  MoveL (T20104) to (112.13, 109.45, 20.1) mm, rotated rx 180 ry 0 rz -180 deg; joints [1.817, 69.838, -35.399, 3.211, -34.481, -2.648]
  Call Extruder 0.01136
  MoveL (T20105) to (122.25, 109.45, 20.1) mm, rotated rx 180 ry 0 rz -180 deg; joints [1.817, 69.838, -35.399, 3.211, -34.481, -2.648]
  Call Extruder 0.00011
  MoveL (T20106) to (122.25, 109.35, 20.1) mm, rotated rx 180 ry 0 rz -180 deg; joints [1.817, 69.838, -35.399, 3.211, -34.481, -2.648]
  Call Extruder 0.01142
  MoveL (T20107) to (112.08, 109.35, 20.1) mm, rotated rx 180 ry 0 rz -180 deg; joints [1.416, 68.674, -33.212, 2.439, -35.486, -1.986]
  Call Extruder 0.00013
  MoveL (T20108) to (112.03, 109.25, 20.1) mm, rotated rx 180 ry 0 rz -180 deg; joints [1.416, 68.674, -33.212, 2.439, -35.486, -1.986]
  Call Extruder 0.01148
  MoveL (T20109) to (122.25, 109.25, 20.1) mm, rotated rx 180 ry 0 rz -180 deg; joints [1.416, 68.674, -33.212, 2.439, -35.486, -1.986]
  Call Extruder 0.00011
  MoveL (T20110) to (122.25, 109.15, 20.1) mm, rotated rx 180 ry 0 rz -180 deg; joints [1.417, 68.506, -32.897, 2.433, -35.633, -1.978]
  Call Extruder 0.01153
  MoveL (T20111) to (111.98, 109.15, 20.1) mm, rotated rx 180 ry 0 rz -180 deg; joints [1.417, 68.506, -32.897, 2.433, -35.633, -1.978]
  Call Extruder 0.00013
  MoveL (T20112) to (111.92, 109.05, 20.1) mm, rotated rx 180 ry 0 rz -180 deg; joints [1.819, 69.662, -35.069, 3.202, -34.636, -2.636]
  Call Extruder 0.01159
  MoveL (T20113) to (122.25, 109.05, 20.1) mm, rotated rx 180 ry 0 rz -180 deg; joints [1.819, 69.662, -35.069, 3.202, -34.636, -2.636]
  Call Extruder 0.00011
  MoveL (T20114) to (122.25, 108.95, 20.1) mm, rotated rx 180 ry 0 rz -180 deg; joints [1.819, 69.662, -35.069, 3.202, -34.636, -2.636]
  Call Extruder 0.01165
  MoveL (T20115) to (111.87, 108.95, 20.1) mm, rotated rx 180 ry 0 rz -180 deg; joints [1.821, 69.488, -34.741, 3.193, -34.789, -2.624]
  Call Extruder 0.00013
  MoveL (T20116) to (111.82, 108.85, 20.1) mm, rotated rx 180 ry 0 rz -180 deg; joints [1.821, 69.488, -34.741, 3.193, -34.789, -2.624]
  Call Extruder 0.01171
  MoveL (T20117) to (122.25, 108.85, 20.1) mm, rotated rx 180 ry 0 rz -180 deg; joints [1.419, 68.339, -32.584, 2.427, -35.78, -1.969]
  Call Extruder 0.00011
  MoveL (T20118) to (122.25, 108.75, 20.1) mm, rotated rx 180 ry 0 rz -180 deg; joints [1.419, 68.339, -32.584, 2.427, -35.78, -1.969]
  Call Extruder 0.01176
  MoveL (T20119) to (111.77, 108.75, 20.1) mm, rotated rx 180 ry 0 rz -180 deg; joints [1.42, 68.174, -32.273, 2.421, -35.925, -1.961]
  Call Extruder 0.00013
  MoveL (T20120) to (111.72, 108.65, 20.1) mm, rotated rx 180 ry 0 rz -180 deg; joints [1.42, 68.174, -32.273, 2.421, -35.925, -1.961]
  Call Extruder 0.01182
  MoveL (T20121) to (122.25, 108.65, 20.1) mm, rotated rx 180 ry 0 rz -180 deg; joints [1.42, 68.174, -32.273, 2.421, -35.925, -1.961]
  Call Extruder 0.00011
  MoveL (T20122) to (122.25, 108.55, 20.1) mm, rotated rx 180 ry 0 rz -180 deg; joints [1.823, 69.314, -34.415, 3.185, -34.941, -2.612]
  Call Extruder 0.01188
  MoveL (T20123) to (111.67, 108.55, 20.1) mm, rotated rx 180 ry 0 rz -180 deg; joints [1.823, 69.314, -34.415, 3.185, -34.941, -2.612]
  Call Extruder 0.00013
  MoveL (T20124) to (111.62, 108.45, 20.1) mm, rotated rx 180 ry 0 rz -180 deg; joints [1.823, 69.314, -34.415, 3.185, -34.941, -2.612]
  Call Extruder 0.01194
  MoveL (T20125) to (122.25, 108.45, 20.1) mm, rotated rx 180 ry 0 rz -180 deg; joints [1.825, 69.142, -34.092, 3.176, -35.092, -2.6]
  Call Extruder 0.00011
  MoveL (T20126) to (122.25, 108.35, 20.1) mm, rotated rx 180 ry 0 rz -180 deg; joints [1.825, 69.142, -34.092, 3.176, -35.092, -2.6]
  Call Extruder 0.01205
  MoveL (T20127) to (111.52, 108.35, 20.1) mm, rotated rx 180 ry 0 rz -180 deg; joints [1.422, 68.009, -31.965, 2.415, -36.069, -1.953]
  Set speed (150.0 mm/s)
  MoveL (T20128) to (111.46, 108.25, 20.1) mm, rotated rx 180 ry 0 rz -180 deg; joints [1.422, 68.009, -31.965, 2.415, -36.069, -1.953]
  Set speed (15.0 mm/s)
  MoveL (T20129) to (111.46, 108.25, 20.1) mm, rotated rx 180 ry 0 rz -180 deg; joints [1.423, 67.846, -31.658, 2.41, -36.212, -1.945]
  Call Extruder 0.01211
  MoveL (T20130) to (122.25, 108.25, 20.1) mm, rotated rx 180 ry 0 rz -180 deg; joints [1.827, 68.971, -33.77, 3.168, -35.242, -2.588]
  Call Extruder 0.00011
  MoveL (T20131) to (122.25, 108.15, 20.1) mm, rotated rx 180 ry 0 rz -180 deg; joints [1.827, 68.971, -33.77, 3.168, -35.242, -2.588]
  Call Extruder 0.00605
  MoveL (T20132) to (116.86, 108.15, 20.1) mm, rotated rx 180 ry 0 rz -180 deg; joints [1.827, 68.971, -33.77, 3.168, -35.242, -2.588]
  Call Extruder 0.00011
  MoveL (T20133) to (116.86, 108.05, 20.1) mm, rotated rx 180 ry 0 rz -180 deg; joints [1.829, 68.801, -33.452, 3.16, -35.391, -2.577]
  Call Extruder 0.00605
  MoveL (T20134) to (122.25, 108.05, 20.1) mm, rotated rx 180 ry 0 rz -180 deg; joints [1.829, 68.801, -33.452, 3.16, -35.391, -2.577]
  Call Extruder 0.00011
  MoveL (T20135) to (122.25, 107.95, 20.1) mm, rotated rx 180 ry 0 rz -180 deg; joints [1.829, 68.801, -33.452, 3.16, -35.391, -2.577]
  Call Extruder 0.00605
  MoveL (T20136) to (116.86, 107.95, 20.1) mm, rotated rx 180 ry 0 rz -180 deg; joints [1.425, 67.684, -31.353, 2.404, -36.355, -1.937]
  Call Extruder 0.00011
  MoveL (T20137) to (116.86, 107.85, 20.1) mm, rotated rx 180 ry 0 rz -180 deg; joints [1.425, 67.684, -31.353, 2.404, -36.355, -1.937]
  Call Extruder 0.00605
  MoveL (T20138) to (122.25, 107.85, 20.1) mm, rotated rx 180 ry 0 rz -180 deg; joints [1.425, 67.684, -31.353, 2.404, -36.355, -1.937]
  Call Extruder 0.00011
  MoveL (T20139) to (122.25, 107.75, 20.1) mm, rotated rx 180 ry 0 rz -180 deg; joints [1.427, 67.522, -31.05, 2.399, -36.496, -1.929]
  Call Extruder 0.00605
  MoveL (T20140) to (116.86, 107.75, 20.1) mm, rotated rx 180 ry 0 rz -180 deg; joints [1.427, 67.522, -31.05, 2.399, -36.496, -1.929]
  Call Extruder 0.00011
  MoveL (T20141) to (116.86, 107.65, 20.1) mm, rotated rx 180 ry 0 rz -180 deg; joints [1.69, 68.237, -32.392, 2.885, -35.88, -2.338]
  Call Extruder 0.00605
  MoveL (T20142) to (122.25, 107.65, 20.1) mm, rotated rx 180 ry 0 rz -180 deg; joints [1.69, 68.237, -32.392, 2.885, -35.88, -2.338]
  Call Extruder 0.00011
  MoveL (T20143) to (122.25, 107.55, 20.1) mm, rotated rx 180 ry 0 rz -180 deg; joints [1.723, 68.157, -32.241, 2.935, -35.951, -2.377]
  Call Extruder 0.00605
  MoveL (T20144) to (116.86, 107.55, 20.1) mm, rotated rx 180 ry 0 rz -180 deg; joints [1.723, 68.157, -32.241, 2.935, -35.951, -2.377]
  Call Extruder 0.00011
  MoveL (T20145) to (116.86, 107.45, 20.1) mm, rotated rx 180 ry 0 rz -180 deg; joints [1.723, 68.157, -32.241, 2.935, -35.951, -2.377]
  Call Extruder 0.00605
  MoveL (T20146) to (122.25, 107.45, 20.1) mm, rotated rx 180 ry 0 rz -180 deg; joints [1.428, 67.362, -30.749, 2.394, -36.637, -1.921]
  Call Extruder 0.00011
  MoveL (T20147) to (122.25, 107.35, 20.1) mm, rotated rx 180 ry 0 rz -180 deg; joints [1.428, 67.362, -30.749, 2.394, -36.637, -1.921]
  Call Extruder 0.00605
  MoveL (T20148) to (116.86, 107.35, 20.1) mm, rotated rx 180 ry 0 rz -180 deg; joints [1.428, 67.362, -30.749, 2.394, -36.637, -1.921]
  Call Extruder 0.00011
  MoveL (T20149) to (116.86, 107.25, 20.1) mm, rotated rx 180 ry 0 rz -180 deg; joints [1.43, 67.202, -30.45, 2.389, -36.777, -1.914]
  Call Extruder 0.00605
  MoveL (T20150) to (122.25, 107.25, 20.1) mm, rotated rx 180 ry 0 rz -180 deg; joints [1.43, 67.202, -30.45, 2.389, -36.777, -1.914]
  Call Extruder 0.00011
  MoveL (T20151) to (122.25, 107.15, 20.1) mm, rotated rx 180 ry 0 rz -180 deg; joints [1.43, 67.202, -30.45, 2.389, -36.777, -1.914]
  Call Extruder 0.00605
  MoveL (T20152) to (116.86, 107.15, 20.1) mm, rotated rx 180 ry 0 rz -180 deg; joints [1.755, 68.077, -32.091, 2.986, -36.023, -2.416]
  Call Extruder 0.00011
  MoveL (T20153) to (116.86, 107.05, 20.1) mm, rotated rx 180 ry 0 rz -180 deg; joints [1.755, 68.077, -32.091, 2.986, -36.023, -2.416]
  Call Extruder 0.00605
  MoveL (T20154) to (122.25, 107.05, 20.1) mm, rotated rx 180 ry 0 rz -180 deg; joints [1.755, 68.077, -32.091, 2.986, -36.023, -2.416]
  Call Extruder 0.00011
  MoveL (T20155) to (122.25, 106.95, 20.1) mm, rotated rx 180 ry 0 rz -180 deg; joints [1.788, 67.998, -31.942, 3.036, -36.093, -2.454]
  Call Extruder 0.00605
  MoveL (T20156) to (116.86, 106.95, 20.1) mm, rotated rx 180 ry 0 rz -180 deg; joints [1.431, 67.044, -30.153, 2.383, -36.915, -1.906]
  Call Extruder 0.00011
  MoveL (T20157) to (116.86, 106.85, 20.1) mm, rotated rx 180 ry 0 rz -180 deg; joints [1.431, 67.044, -30.153, 2.383, -36.915, -1.906]
  Call Extruder 0.00605
  MoveL (T20158) to (122.25, 106.85, 20.1) mm, rotated rx 180 ry 0 rz -180 deg; joints [1.431, 67.044, -30.153, 2.383, -36.915, -1.906]
  Call Extruder 0.00011
  MoveL (T20159) to (122.25, 106.75, 20.1) mm, rotated rx 180 ry 0 rz -180 deg; joints [1.433, 66.887, -29.857, 2.379, -37.053, -1.899]
  Call Extruder 0.00605
  MoveL (T20160) to (116.86, 106.75, 20.1) mm, rotated rx 180 ry 0 rz -180 deg; joints [1.433, 66.887, -29.857, 2.379, -37.053, -1.899]
  Call Extruder 0.00011
  MoveL (T20161) to (116.86, 106.65, 20.1) mm, rotated rx 180 ry 0 rz -180 deg; joints [1.433, 66.887, -29.857, 2.379, -37.053, -1.899]
  Call Extruder 0.00605
  MoveL (T20162) to (122.25, 106.65, 20.1) mm, rotated rx 180 ry 0 rz -180 deg; joints [1.821, 67.918, -31.794, 3.087, -36.164, -2.493]
  Call Extruder 0.00011
  MoveL (T20163) to (122.25, 106.55, 20.1) mm, rotated rx 180 ry 0 rz -180 deg; joints [1.821, 67.918, -31.794, 3.087, -36.164, -2.493]
  Call Extruder 0.00605
  MoveL (T20164) to (116.86, 106.55, 20.1) mm, rotated rx 180 ry 0 rz -180 deg; joints [1.838, 67.876, -31.714, 3.114, -36.202, -2.513]
  Call Extruder 0.00011
  MoveL (T20165) to (116.86, 106.45, 20.1) mm, rotated rx 180 ry 0 rz -180 deg; joints [1.838, 67.876, -31.714, 3.114, -36.202, -2.513]
  Call Extruder 0.00605
  MoveL (T20166) to (122.25, 106.45, 20.1) mm, rotated rx 180 ry 0 rz -180 deg; joints [1.838, 67.876, -31.714, 3.114, -36.202, -2.513]
  Call Extruder 0.00011
  MoveL (T20167) to (122.25, 106.35, 20.1) mm, rotated rx 180 ry 0 rz -180 deg; joints [1.838, 67.876, -31.714, 3.114, -36.202, -2.513]
  Call Extruder 0.0061
  MoveL (T20168) to (116.82, 106.35, 20.1) mm, rotated rx 180 ry 0 rz -180 deg; joints [1.838, 67.876, -31.714, 3.114, -36.202, -2.513]
  Set speed (45.0 mm/s)
  Call Extruder -1.6
  MoveL (T20169) to (116.82, 106.35, 20.1) mm, rotated rx 180 ry 0 rz -180 deg; joints [1.838, 67.876, -31.714, 3.114, -36.202, -2.513]
  Set speed (120.0 mm/s)
  MoveL (T20170) to (116.82, 106.35, 20.1) mm, rotated rx 180 ry 0 rz -180 deg; joints [1.841, 67.862, -31.688, 3.117, -36.215, -2.516]
  Call Extruder -0.38
  MoveL (T20171) to (117.88, 106.35, 20.1) mm, rotated rx 180 ry 0 rz -180 deg; joints [1.842, 67.806, -31.584, 3.115, -36.263, -2.512]
  Set speed (45.0 mm/s)
  Call Extruder -0.02
  MoveL (T20172) to (117.88, 106.35, 20.1) mm, rotated rx 180 ry 0 rz -180 deg; joints [1.842, 67.806, -31.584, 3.115, -36.263, -2.512]
  Set speed (150.0 mm/s)
  MoveL (T20173) to (117.88, 106.35, 22.1) mm, rotated rx 180 ry 0 rz -180 deg; joints [1.435, 66.73, -29.563, 2.374, -37.191, -1.891]
  MoveL (T20174) to (108.7, 118.95, 22.1) mm, rotated rx 180 ry 0 rz -180 deg; joints [1.435, 66.73, -29.563, 2.374, -37.191, -1.891]
  MoveL (T20175) to (108.7, 118.95, 20.1) mm, rotated rx 180 ry 0 rz -180 deg; joints [1.435, 66.73, -29.563, 2.374, -37.191, -1.891]
  Set speed (40.0 mm/s)
  Call Extruder 2.0
  MoveL (T20176) to (108.7, 118.95, 20.1) mm, rotated rx 180 ry 0 rz -180 deg; joints [1.436, 66.574, -29.271, 2.369, -37.327, -1.884]
  Set speed (15.0 mm/s)
  MoveL (T20177) to (108.7, 118.95, 20.1) mm, rotated rx 180 ry 0 rz -180 deg; joints [1.436, 66.574, -29.271, 2.369, -37.327, -1.884]
  Call Extruder 0.00668
  MoveL (T20178) to (102.75, 118.95, 20.1) mm, rotated rx 180 ry 0 rz -180 deg; joints [1.436, 66.574, -29.271, 2.369, -37.327, -1.884]
  Call Extruder 0.00011
  MoveL (T20179) to (102.75, 118.85, 20.1) mm, rotated rx 180 ry 0 rz -180 deg; joints [1.844, 67.644, -31.28, 3.107, -36.405, -2.502]
  Call Extruder 0.00663
  MoveL (T20180) to (108.66, 118.85, 20.1) mm, rotated rx 180 ry 0 rz -180 deg; joints [1.844, 67.644, -31.28, 3.107, -36.405, -2.502]
  Call Extruder 0.00011
  MoveL (T20181) to (108.66, 118.75, 20.1) mm, rotated rx 180 ry 0 rz -180 deg; joints [1.846, 67.483, -30.977, 3.101, -36.546, -2.492]
  Call Extruder 0.00663
  MoveL (T20182) to (102.75, 118.75, 20.1) mm, rotated rx 180 ry 0 rz -180 deg; joints [1.438, 66.419, -28.98, 2.364, -37.463, -1.877]
  Call Extruder 0.00011
  MoveL (T20183) to (102.75, 118.65, 20.1) mm, rotated rx 180 ry 0 rz -180 deg; joints [1.438, 66.419, -28.98, 2.364, -37.463, -1.877]
  Call Extruder 0.00663
  MoveL (T20184) to (108.66, 118.65, 20.1) mm, rotated rx 180 ry 0 rz -180 deg; joints [1.439, 66.266, -28.692, 2.36, -37.597, -1.87]
  Call Extruder 0.00011
  MoveL (T20185) to (108.66, 118.55, 20.1) mm, rotated rx 180 ry 0 rz -180 deg; joints [1.439, 66.266, -28.692, 2.36, -37.597, -1.87]
  Call Extruder 0.00663
  MoveL (T20186) to (102.75, 118.55, 20.1) mm, rotated rx 180 ry 0 rz -180 deg; joints [1.439, 66.266, -28.692, 2.36, -37.597, -1.87]
  Call Extruder 0.00011
  MoveL (T20187) to (102.75, 118.45, 20.1) mm, rotated rx 180 ry 0 rz -180 deg; joints [1.439, 66.266, -28.692, 2.36, -37.597, -1.87]
  Call Extruder 0.00663
  MoveL (T20188) to (108.66, 118.45, 20.1) mm, rotated rx 180 ry 0 rz -180 deg; joints [1.848, 67.323, -30.677, 3.094, -36.687, -2.482]
  Call Extruder 0.00011
  MoveL (T20189) to (108.66, 118.35, 20.1) mm, rotated rx 180 ry 0 rz -180 deg; joints [1.848, 67.323, -30.677, 3.094, -36.687, -2.482]
  Call Extruder 0.00663
  MoveL (T20190) to (102.75, 118.35, 20.1) mm, rotated rx 180 ry 0 rz -180 deg; joints [1.848, 67.323, -30.677, 3.094, -36.687, -2.482]
  Call Extruder 0.00011
  MoveL (T20191) to (102.75, 118.25, 20.1) mm, rotated rx 180 ry 0 rz -180 deg; joints [1.85, 67.164, -30.378, 3.087, -36.826, -2.472]
  Call Extruder 0.00663
  MoveL (T20192) to (108.66, 118.25, 20.1) mm, rotated rx 180 ry 0 rz -180 deg; joints [1.85, 67.164, -30.378, 3.087, -36.826, -2.472]
  Call Extruder 0.00011
  MoveL (T20193) to (108.66, 118.15, 20.1) mm, rotated rx 180 ry 0 rz -180 deg; joints [1.85, 67.164, -30.378, 3.087, -36.826, -2.472]
  Call Extruder 0.00663
  MoveL (T20194) to (102.75, 118.15, 20.1) mm, rotated rx 180 ry 0 rz -180 deg; joints [1.456, 66.151, -28.477, 2.382, -37.698, -1.885]
  Call Extruder 0.00011
  MoveL (T20195) to (102.75, 118.05, 20.1) mm, rotated rx 180 ry 0 rz -180 deg; joints [1.456, 66.151, -28.477, 2.382, -37.698, -1.885]
  Call Extruder 0.00663
  MoveL (T20196) to (108.66, 118.05, 20.1) mm, rotated rx 180 ry 0 rz -180 deg; joints [1.456, 66.151, -28.477, 2.382, -37.698, -1.885]
  Call Extruder 0.00011
  MoveL (T20197) to (108.66, 117.95, 20.1) mm, rotated rx 180 ry 0 rz -180 deg; joints [1.521, 66.155, -28.484, 2.488, -37.697, -1.969]
  Call Extruder 0.00663
  MoveL (T20198) to (102.75, 117.95, 20.1) mm, rotated rx 180 ry 0 rz -180 deg; joints [1.521, 66.155, -28.484, 2.488, -37.697, -1.969]
  Call Extruder 0.00011
  MoveL (T20199) to (102.75, 117.85, 20.1) mm, rotated rx 180 ry 0 rz -180 deg; joints [1.521, 66.155, -28.484, 2.488, -37.697, -1.969]
  Call Extruder 0.00663
  MoveL (T20200) to (108.66, 117.85, 20.1) mm, rotated rx 180 ry 0 rz -180 deg; joints [1.852, 67.006, -30.081, 3.081, -36.965, -2.462]
  Call Extruder 0.00011
  MoveL (T20201) to (108.66, 117.75, 20.1) mm, rotated rx 180 ry 0 rz -180 deg; joints [1.852, 67.006, -30.081, 3.081, -36.965, -2.462]
  Call Extruder 0.00663
  MoveL (T20202) to (102.75, 117.75, 20.1) mm, rotated rx 180 ry 0 rz -180 deg; joints [1.852, 67.006, -30.081, 3.081, -36.965, -2.462]
  Call Extruder 0.00011
  MoveL (T20203) to (102.75, 117.65, 20.1) mm, rotated rx 180 ry 0 rz -180 deg; joints [1.854, 66.849, -29.786, 3.074, -37.102, -2.453]
  Call Extruder 0.00663
  MoveL (T20204) to (108.66, 117.65, 20.1) mm, rotated rx 180 ry 0 rz -180 deg; joints [1.854, 66.849, -29.786, 3.074, -37.102, -2.453]
  Call Extruder 0.00011
  MoveL (T20205) to (108.66, 117.55, 20.1) mm, rotated rx 180 ry 0 rz -180 deg; joints [1.585, 66.159, -28.493, 2.593, -37.695, -2.052]
  Call Extruder 0.00663
  MoveL (T20206) to (102.75, 117.55, 20.1) mm, rotated rx 180 ry 0 rz -180 deg; joints [1.585, 66.159, -28.493, 2.593, -37.695, -2.052]
  Call Extruder 0.00011
  MoveL (T20207) to (102.75, 117.45, 20.1) mm, rotated rx 180 ry 0 rz -180 deg; joints [1.585, 66.159, -28.493, 2.593, -37.695, -2.052]
  Call Extruder 0.00663
  MoveL (T20208) to (108.66, 117.45, 20.1) mm, rotated rx 180 ry 0 rz -180 deg; joints [1.647, 66.164, -28.501, 2.694, -37.694, -2.133]
  Call Extruder 0.00011
  MoveL (T20209) to (108.66, 117.35, 20.1) mm, rotated rx 180 ry 0 rz -180 deg; joints [1.647, 66.164, -28.501, 2.694, -37.694, -2.133]
  Call Extruder 0.00663
  MoveL (T20210) to (102.75, 117.35, 20.1) mm, rotated rx 180 ry 0 rz -180 deg; joints [1.647, 66.164, -28.501, 2.694, -37.694, -2.133]
  Call Extruder 0.00011
  MoveL (T20211) to (102.75, 117.25, 20.1) mm, rotated rx 180 ry 0 rz -180 deg; joints [1.651, 66.168, -28.508, 2.701, -37.69, -2.138]
  Call Extruder 0.00663
  MoveL (T20212) to (108.66, 117.25, 20.1) mm, rotated rx 180 ry 0 rz -180 deg; joints [1.651, 66.168, -28.508, 2.701, -37.69, -2.138]
  Call Extruder 0.00011
  MoveL (T20213) to (108.66, 117.15, 20.1) mm, rotated rx 180 ry 0 rz -180 deg; joints [1.875, 66.742, -29.586, 3.103, -37.197, -2.472]
  Call Extruder 0.00663
  MoveL (T20214) to (102.75, 117.15, 20.1) mm, rotated rx 180 ry 0 rz -180 deg; joints [1.875, 66.742, -29.586, 3.103, -37.197, -2.472]
  Call Extruder 0.00011
  MoveL (T20215) to (102.75, 117.05, 20.1) mm, rotated rx 180 ry 0 rz -180 deg; joints [1.875, 66.742, -29.586, 3.103, -37.197, -2.472]
  Call Extruder 0.0123
  MoveL (T20216) to (113.7, 117.05, 20.1) mm, rotated rx 180 ry 0 rz -180 deg; joints [1.875, 66.742, -29.586, 3.103, -37.197, -2.472]
  Call Extruder 0.00013
  MoveL (T20217) to (113.65, 116.95, 20.1) mm, rotated rx 180 ry 0 rz -180 deg; joints [1.875, 66.742, -29.586, 3.103, -37.197, -2.472]
  Call Extruder 0.01224
  MoveL (T20218) to (102.75, 116.95, 20.1) mm, rotated rx 180 ry 0 rz -180 deg; joints [1.875, 66.742, -29.586, 3.103, -37.197, -2.472]
  Call Extruder 0.00011
  MoveL (T20219) to (102.75, 116.85, 20.1) mm, rotated rx 180 ry 0 rz -180 deg; joints [1.875, 66.742, -29.586, 3.103, -37.197, -2.472]
  Call Extruder 0.01218
  MoveL (T20220) to (113.6, 116.85, 20.1) mm, rotated rx 180 ry 0 rz -180 deg; joints [1.796, 66.538, -29.203, 2.96, -37.372, -2.353]
  Call Extruder 0.00013
  MoveL (T20221) to (113.55, 116.75, 20.1) mm, rotated rx 180 ry 0 rz -180 deg; joints [1.796, 66.538, -29.203, 2.96, -37.372, -2.353]
  Call Extruder 0.01213
  MoveL (T20222) to (102.75, 116.75, 20.1) mm, rotated rx 180 ry 0 rz -180 deg; joints [1.796, 66.538, -29.203, 2.96, -37.372, -2.353]
  Call Extruder 0.00011
  MoveL (T20223) to (102.75, 116.65, 20.1) mm, rotated rx 180 ry 0 rz -180 deg; joints [1.796, 66.538, -29.203, 2.96, -37.372, -2.353]
  Call Extruder 0.01207
  MoveL (T20224) to (113.5, 116.65, 20.1) mm, rotated rx 180 ry 0 rz -180 deg; joints [1.796, 66.538, -29.203, 2.96, -37.372, -2.353]
  Call Extruder 0.00013
  MoveL (T20225) to (113.45, 116.55, 20.1) mm, rotated rx 180 ry 0 rz -180 deg; joints [1.796, 66.538, -29.203, 2.96, -37.372, -2.353]
  Call Extruder 0.01201
  MoveL (T20226) to (102.75, 116.55, 20.1) mm, rotated rx 180 ry 0 rz -180 deg; joints [1.796, 66.538, -29.203, 2.96, -37.372, -2.353]
  Call Extruder 0.00011
  MoveL (T20227) to (102.75, 116.45, 20.1) mm, rotated rx 180 ry 0 rz -180 deg; joints [1.796, 66.538, -29.203, 2.96, -37.372, -2.353]
  Call Extruder 0.01195
  MoveL (T20228) to (113.4, 116.45, 20.1) mm, rotated rx 180 ry 0 rz -180 deg; joints [1.796, 66.538, -29.203, 2.96, -37.372, -2.353]
  Call Extruder 0.00013
  MoveL (T20229) to (113.35, 116.35, 20.1) mm, rotated rx 180 ry 0 rz -180 deg; joints [1.796, 66.303, -29.168, 2.974, -37.173, -2.37]
  Call Extruder 0.0119
  MoveL (T20230) to (102.75, 116.35, 20.1) mm, rotated rx 180 ry 0 rz -180 deg; joints [3.301, 66.633, -29.785, 5.494, -36.974, -4.394]
  Call Extruder 0.00011
  MoveL (T20231) to (102.75, 116.25, 20.1) mm, rotated rx 180 ry 0 rz -180 deg; joints [3.301, 66.867, -29.821, 5.469, -37.172, -4.362]
  Call Extruder 0.01184
  MoveL (T20232) to (113.3, 116.25, 20.1) mm, rotated rx 180 ry 0 rz -180 deg; joints [3.301, 66.867, -29.821, 5.469, -37.172, -4.362]
  Call Extruder 0.00013
  MoveL (T20233) to (113.25, 116.15, 20.1) mm, rotated rx 180 ry 0 rz -180 deg; joints [3.301, 66.867, -29.821, 5.469, -37.172, -4.362]
  Call Extruder 0.01178
  MoveL (T20234) to (102.75, 116.15, 20.1) mm, rotated rx 180 ry 0 rz -180 deg; joints [3.301, 66.867, -29.821, 5.469, -37.172, -4.362]
  Call Extruder 0.00011
  MoveL (T20235) to (102.75, 116.05, 20.1) mm, rotated rx 180 ry 0 rz -180 deg; joints [3.301, 66.867, -29.821, 5.469, -37.172, -4.362]
  Call Extruder 0.01173
  MoveL (T20236) to (113.19, 116.05, 20.1) mm, rotated rx 180 ry 0 rz -180 deg; joints [3.301, 66.867, -29.821, 5.469, -37.172, -4.362]
  Call Extruder 0.00013
  MoveL (T20237) to (113.14, 115.95, 20.1) mm, rotated rx 180 ry 0 rz -180 deg; joints [3.301, 66.867, -29.821, 5.469, -37.172, -4.362]
  Call Extruder 0.01167
  MoveL (T20238) to (102.75, 115.95, 20.1) mm, rotated rx 180 ry 0 rz -180 deg; joints [3.301, 66.867, -29.821, 5.469, -37.172, -4.362]
  Call Extruder 0.00011
  MoveL (T20239) to (102.75, 115.85, 20.1) mm, rotated rx 180 ry 0 rz -180 deg; joints [3.301, 66.867, -29.821, 5.469, -37.172, -4.362]
  Call Extruder 0.01161
  MoveL (T20240) to (113.09, 115.85, 20.1) mm, rotated rx 180 ry 0 rz -180 deg; joints [3.301, 66.867, -29.821, 5.469, -37.172, -4.362]
  Call Extruder 0.00013
  MoveL (T20241) to (113.04, 115.75, 20.1) mm, rotated rx 180 ry 0 rz -180 deg; joints [3.301, 66.867, -29.821, 5.469, -37.172, -4.362]
  Call Extruder 0.01155
  MoveL (T20242) to (102.75, 115.75, 20.1) mm, rotated rx 180 ry 0 rz -180 deg; joints [3.316, 66.23, -28.624, 5.424, -37.73, -4.295]
  Call Extruder 0.00011
  MoveL (T20243) to (102.75, 115.65, 20.1) mm, rotated rx 180 ry 0 rz -180 deg; joints [3.316, 66.23, -28.624, 5.424, -37.73, -4.295]
  Call Extruder 0.0115
  MoveL (T20244) to (112.99, 115.65, 20.1) mm, rotated rx 180 ry 0 rz -180 deg; joints [1.863, 69.649, -35.043, 3.277, -34.65, -2.697]
  Call Extruder 0.00013
  MoveL (T20245) to (112.94, 115.55, 20.1) mm, rotated rx 180 ry 0 rz -180 deg; joints [1.863, 69.649, -35.043, 3.277, -34.65, -2.697]
  Call Extruder 0.01144
  MoveL (T20246) to (102.75, 115.55, 20.1) mm, rotated rx 180 ry 0 rz -180 deg; joints [1.863, 69.649, -35.043, 3.277, -34.65, -2.697]
  Call Extruder 0.00011
  MoveL (T20247) to (102.75, 115.45, 20.1) mm, rotated rx 180 ry 0 rz -180 deg; joints [1.863, 69.649, -35.043, 3.277, -34.65, -2.697]
  Call Extruder 0.01138
  MoveL (T20248) to (112.89, 115.45, 20.1) mm, rotated rx 180 ry 0 rz -180 deg; joints [1.861, 69.801, -35.328, 3.285, -34.517, -2.708]
  Call Extruder 0.00013
  MoveL (T20249) to (112.84, 115.35, 20.1) mm, rotated rx 180 ry 0 rz -180 deg; joints [1.861, 69.801, -35.328, 3.285, -34.517, -2.708]
  Call Extruder 0.01132
  MoveL (T20250) to (102.75, 115.35, 20.1) mm, rotated rx 180 ry 0 rz -180 deg; joints [1.861, 69.801, -35.328, 3.285, -34.517, -2.708]
  Call Extruder 0.00011
  MoveL (T20251) to (102.75, 115.25, 20.1) mm, rotated rx 180 ry 0 rz -180 deg; joints [1.915, 69.963, -35.633, 3.392, -34.377, -2.801]
  Call Extruder 0.01127
  MoveL (T20252) to (112.79, 115.25, 20.1) mm, rotated rx 180 ry 0 rz -180 deg; joints [1.915, 69.963, -35.633, 3.392, -34.377, -2.801]
  Call Extruder 0.00013
  MoveL (T20253) to (112.74, 115.15, 20.1) mm, rotated rx 180 ry 0 rz -180 deg; joints [1.915, 69.963, -35.633, 3.392, -34.377, -2.801]
  Call Extruder 0.01121
  MoveL (T20254) to (102.75, 115.15, 20.1) mm, rotated rx 180 ry 0 rz -180 deg; joints [1.915, 69.963, -35.633, 3.392, -34.377, -2.801]
  Call Extruder 0.00011
  MoveL (T20255) to (102.75, 115.05, 20.1) mm, rotated rx 180 ry 0 rz -180 deg; joints [1.803, 70.262, -36.195, 3.216, -34.109, -2.664]
  Call Extruder 0.01115
  MoveL (T20256) to (112.69, 115.05, 20.1) mm, rotated rx 180 ry 0 rz -180 deg; joints [1.794, 70.323, -36.308, 3.204, -34.056, -2.655]
  Call Extruder 0.00013
  MoveL (T20257) to (112.63, 114.95, 20.1) mm, rotated rx 180 ry 0 rz -180 deg; joints [1.794, 70.323, -36.308, 3.204, -34.056, -2.655]
  Call Extruder 0.0111
  MoveL (T20258) to (102.75, 114.95, 20.1) mm, rotated rx 180 ry 0 rz -180 deg; joints [1.787, 70.951, -37.489, 3.238, -33.504, -2.701]
  Call Extruder 0.00011
  MoveL (T20259) to (102.75, 114.85, 20.1) mm, rotated rx 180 ry 0 rz -180 deg; joints [1.787, 70.951, -37.489, 3.238, -33.504, -2.701]
  Call Extruder 0.01104
  MoveL (T20260) to (112.58, 114.85, 20.1) mm, rotated rx 180 ry 0 rz -180 deg; joints [1.763, 70.949, -37.485, 3.195, -33.505, -2.665]
  Call Extruder 0.00013
  MoveL (T20261) to (112.53, 114.75, 20.1) mm, rotated rx 180 ry 0 rz -180 deg; joints [1.763, 70.949, -37.485, 3.195, -33.505, -2.665]
  Call Extruder 0.01098
  MoveL (T20262) to (102.75, 114.75, 20.1) mm, rotated rx 180 ry 0 rz -180 deg; joints [1.763, 70.949, -37.485, 3.195, -33.505, -2.665]
  Call Extruder 0.00011
  MoveL (T20263) to (102.75, 114.65, 20.1) mm, rotated rx 180 ry 0 rz -180 deg; joints [1.659, 70.622, -36.871, 2.983, -33.787, -2.48]
  Call Extruder 0.01092
  MoveL (T20264) to (112.48, 114.65, 20.1) mm, rotated rx 180 ry 0 rz -180 deg; joints [1.659, 70.622, -36.871, 2.983, -33.787, -2.48]
  Call Extruder 0.00013
  MoveL (T20265) to (112.43, 114.55, 20.1) mm, rotated rx 180 ry 0 rz -180 deg; joints [1.659, 70.622, -36.871, 2.983, -33.787, -2.48]
  Call Extruder 0.01087
  MoveL (T20266) to (102.75, 114.55, 20.1) mm, rotated rx 180 ry 0 rz -180 deg; joints [1.628, 70.707, -37.03, 2.934, -33.711, -2.441]
  Call Extruder 0.00011
  MoveL (T20267) to (102.75, 114.45, 20.1) mm, rotated rx 180 ry 0 rz -180 deg; joints [1.628, 70.707, -37.03, 2.934, -33.711, -2.441]
  Call Extruder 0.01081
  MoveL (T20268) to (112.38, 114.45, 20.1) mm, rotated rx 180 ry 0 rz -180 deg; joints [1.628, 70.707, -37.03, 2.934, -33.711, -2.441]
  Call Extruder 0.00013
  MoveL (T20269) to (112.33, 114.35, 20.1) mm, rotated rx 180 ry 0 rz -180 deg; joints [1.607, 70.731, -37.075, 2.897, -33.689, -2.411]
  Call Extruder 0.01075
  MoveL (T20270) to (102.75, 114.35, 20.1) mm, rotated rx 180 ry 0 rz -180 deg; joints [1.607, 70.731, -37.075, 2.897, -33.689, -2.411]
  Call Extruder 0.00011
  MoveL (T20271) to (102.75, 114.25, 20.1) mm, rotated rx 180 ry 0 rz -180 deg; joints [1.607, 70.731, -37.075, 2.897, -33.689, -2.411]
  Call Extruder 0.01069
  MoveL (T20272) to (112.28, 114.25, 20.1) mm, rotated rx 180 ry 0 rz -180 deg; joints [1.467, 70.72, -37.055, 2.644, -33.693, -2.201]
  Call Extruder 0.00013
  MoveL (T20273) to (112.23, 114.15, 20.1) mm, rotated rx 180 ry 0 rz -180 deg; joints [1.467, 70.72, -37.055, 2.644, -33.693, -2.201]
  Call Extruder 0.01064
  MoveL (T20274) to (102.75, 114.15, 20.1) mm, rotated rx 180 ry 0 rz -180 deg; joints [1.467, 70.72, -37.055, 2.644, -33.693, -2.201]
  Call Extruder 0.00011
  MoveL (T20275) to (102.75, 114.05, 20.1) mm, rotated rx 180 ry 0 rz -180 deg; joints [1.467, 70.72, -37.055, 2.644, -33.693, -2.201]
  Call Extruder 0.01058
  MoveL (T20276) to (112.17, 114.05, 20.1) mm, rotated rx 180 ry 0 rz -180 deg; joints [1.396, 70.919, -37.429, 2.529, -33.516, -2.109]
  Call Extruder 0.00013
  MoveL (T20277) to (112.12, 113.95, 20.1) mm, rotated rx 180 ry 0 rz -180 deg; joints [1.396, 70.919, -37.429, 2.529, -33.516, -2.109]
  Call Extruder 0.01052
  MoveL (T20278) to (102.75, 113.95, 20.1) mm, rotated rx 180 ry 0 rz -180 deg; joints [1.396, 70.919, -37.429, 2.529, -33.516, -2.109]
  Call Extruder 0.00011
  MoveL (T20279) to (102.75, 113.85, 20.1) mm, rotated rx 180 ry 0 rz -180 deg; joints [1.652, 70.939, -37.467, 2.994, -33.509, -2.497]
  Call Extruder 0.01047
  MoveL (T20280) to (112.07, 113.85, 20.1) mm, rotated rx 180 ry 0 rz -180 deg; joints [1.652, 70.939, -37.467, 2.994, -33.509, -2.497]
  Call Extruder 0.00013
  MoveL (T20281) to (112.02, 113.75, 20.1) mm, rotated rx 180 ry 0 rz -180 deg; joints [1.652, 70.939, -37.467, 2.994, -33.509, -2.497]
  Call Extruder 0.01041
  MoveL (T20282) to (102.75, 113.75, 20.1) mm, rotated rx 180 ry 0 rz -180 deg; joints [1.652, 70.939, -37.467, 2.994, -33.509, -2.497]
  Call Extruder 0.00011
  MoveL (T20283) to (102.75, 113.65, 20.1) mm, rotated rx 180 ry 0 rz -180 deg; joints [1.652, 70.939, -37.467, 2.994, -33.509, -2.497]
  Call Extruder 0.01035
  MoveL (T20284) to (111.97, 113.65, 20.1) mm, rotated rx 180 ry 0 rz -180 deg; joints [1.652, 70.939, -37.467, 2.994, -33.509, -2.497]
  Call Extruder 0.00013
  MoveL (T20285) to (111.92, 113.55, 20.1) mm, rotated rx 180 ry 0 rz -180 deg; joints [1.652, 70.939, -37.467, 2.994, -33.509, -2.497]
  Call Extruder 0.01029
  MoveL (T20286) to (102.75, 113.55, 20.1) mm, rotated rx 180 ry 0 rz -180 deg; joints [1.652, 70.939, -37.467, 2.994, -33.509, -2.497]
  Call Extruder 0.00011
  MoveL (T20287) to (102.75, 113.45, 20.1) mm, rotated rx 180 ry 0 rz -180 deg; joints [1.54, 70.93, -37.449, 2.791, -33.512, -2.327]
  Call Extruder 0.01024
  MoveL (T20288) to (111.87, 113.45, 20.1) mm, rotated rx 180 ry 0 rz -180 deg; joints [1.54, 70.93, -37.449, 2.791, -33.512, -2.327]
  Call Extruder 0.00013
  MoveL (T20289) to (111.82, 113.35, 20.1) mm, rotated rx 180 ry 0 rz -180 deg; joints [1.54, 70.93, -37.449, 2.791, -33.512, -2.327]
  Call Extruder 0.01018
  MoveL (T20290) to (102.75, 113.35, 20.1) mm, rotated rx 180 ry 0 rz -180 deg; joints [1.54, 70.93, -37.449, 2.791, -33.512, -2.327]
  Call Extruder 0.00011
  MoveL (T20291) to (102.75, 113.25, 20.1) mm, rotated rx 180 ry 0 rz -180 deg; joints [1.54, 70.93, -37.449, 2.791, -33.512, -2.327]
  Call Extruder 0.01012
  MoveL (T20292) to (111.77, 113.25, 20.1) mm, rotated rx 180 ry 0 rz -180 deg; joints [1.54, 70.93, -37.449, 2.791, -33.512, -2.327]
  Call Extruder 0.00013
  MoveL (T20293) to (111.72, 113.15, 20.1) mm, rotated rx 180 ry 0 rz -180 deg; joints [1.54, 70.93, -37.449, 2.791, -33.512, -2.327]
  Call Extruder 0.01006
  MoveL (T20294) to (102.75, 113.15, 20.1) mm, rotated rx 180 ry 0 rz -180 deg; joints [1.54, 70.93, -37.449, 2.791, -33.512, -2.327]
  Call Extruder 0.00011
  MoveL (T20295) to (102.75, 113.05, 20.1) mm, rotated rx 180 ry 0 rz -180 deg; joints [1.54, 70.93, -37.449, 2.791, -33.512, -2.327]
  Call Extruder 0.01001
  MoveL (T20296) to (111.67, 113.05, 20.1) mm, rotated rx 180 ry 0 rz -180 deg; joints [1.407, 65.935, -28.477, 2.313, -37.48, -1.836]
  Call Extruder 0.00013
  MoveL (T20297) to (111.61, 112.95, 20.1) mm, rotated rx 180 ry 0 rz -180 deg; joints [1.407, 66.146, -28.509, 2.304, -37.66, -1.824]
  Call Extruder 0.00995
  MoveL (T20298) to (102.75, 112.95, 20.1) mm, rotated rx 180 ry 0 rz -180 deg; joints [1.407, 66.146, -28.509, 2.304, -37.66, -1.824]
  Call Extruder 0.00011
  MoveL (T20299) to (102.75, 112.85, 20.1) mm, rotated rx 180 ry 0 rz -180 deg; joints [1.407, 66.146, -28.509, 2.304, -37.66, -1.824]
  Call Extruder 0.00989
  MoveL (T20300) to (111.56, 112.85, 20.1) mm, rotated rx 180 ry 0 rz -180 deg; joints [1.407, 66.146, -28.509, 2.304, -37.66, -1.824]
  Call Extruder 0.00013
  MoveL (T20301) to (111.51, 112.75, 20.1) mm, rotated rx 180 ry 0 rz -180 deg; joints [1.407, 66.146, -28.509, 2.304, -37.66, -1.824]
  Call Extruder 0.00984
  MoveL (T20302) to (102.75, 112.75, 20.1) mm, rotated rx 180 ry 0 rz -180 deg; joints [1.407, 66.146, -28.509, 2.304, -37.66, -1.824]
  Call Extruder 0.00011
  MoveL (T20303) to (102.75, 112.65, 20.1) mm, rotated rx 180 ry 0 rz -180 deg; joints [1.407, 66.146, -28.509, 2.304, -37.66, -1.824]
  Call Extruder 0.00978
  MoveL (T20304) to (111.46, 112.65, 20.1) mm, rotated rx 180 ry 0 rz -180 deg; joints [1.363, 70.989, -37.599, 2.476, -33.414, -2.067]
  Call Extruder 0.00013
  MoveL (T20305) to (111.41, 112.55, 20.1) mm, rotated rx 180 ry 0 rz -180 deg; joints [1.363, 70.989, -37.599, 2.476, -33.414, -2.067]
  Call Extruder 0.00972
  MoveL (T20306) to (102.75, 112.55, 20.1) mm, rotated rx 180 ry 0 rz -180 deg; joints [1.363, 70.989, -37.599, 2.476, -33.414, -2.067]
  Call Extruder 0.00011
  MoveL (T20307) to (102.75, 112.45, 20.1) mm, rotated rx 180 ry 0 rz -180 deg; joints [3.241, 71.216, -38.026, 5.907, -33.33, -4.94]
  Call Extruder 0.00966
  MoveL (T20308) to (111.36, 112.45, 20.1) mm, rotated rx 180 ry 0 rz -180 deg; joints [3.241, 71.216, -38.026, 5.907, -33.33, -4.94]
  Call Extruder 0.00013
  MoveL (T20309) to (111.31, 112.35, 20.1) mm, rotated rx 180 ry 0 rz -180 deg; joints [3.241, 71.216, -38.026, 5.907, -33.33, -4.94]
  Call Extruder 0.00961
  MoveL (T20310) to (102.75, 112.35, 20.1) mm, rotated rx 180 ry 0 rz -180 deg; joints [3.351, 66.132, -28.482, 5.476, -37.777, -4.333]
  Call Extruder 0.00011
  MoveL (T20311) to (102.75, 112.25, 20.1) mm, rotated rx 180 ry 0 rz -180 deg; joints [3.351, 66.132, -28.482, 5.476, -37.777, -4.333]
  Call Extruder 0.00955
  MoveL (T20312) to (111.26, 112.25, 20.1) mm, rotated rx 180 ry 0 rz -180 deg; joints [1.409, 65.941, -28.123, 2.298, -37.84, -1.815]
  Call Extruder 0.00013
  MoveL (T20313) to (111.21, 112.15, 20.1) mm, rotated rx 180 ry 0 rz -180 deg; joints [1.409, 65.941, -28.123, 2.298, -37.84, -1.815]
  Call Extruder 0.00949
  MoveL (T20314) to (102.75, 112.15, 20.1) mm, rotated rx 180 ry 0 rz -180 deg; joints [1.407, 66.131, -28.479, 2.303, -37.674, -1.823]
  Call Extruder 0.00011
  MoveL (T20315) to (102.75, 112.05, 20.1) mm, rotated rx 180 ry 0 rz -180 deg; joints [1.407, 66.131, -28.479, 2.303, -37.674, -1.823]
  Call Extruder 0.00943
  MoveL (T20316) to (111.16, 112.05, 20.1) mm, rotated rx 180 ry 0 rz -180 deg; joints [1.365, 65.936, -28.115, 2.226, -37.842, -1.758]
  Call Extruder 0.00013
  MoveL (T20317) to (111.1, 111.95, 20.1) mm, rotated rx 180 ry 0 rz -180 deg; joints [1.365, 65.936, -28.115, 2.226, -37.842, -1.758]
  Call Extruder 0.00938
  MoveL (T20318) to (102.75, 111.95, 20.1) mm, rotated rx 180 ry 0 rz -180 deg; joints [1.365, 65.936, -28.115, 2.226, -37.842, -1.758]
  Call Extruder 0.00011
  MoveL (T20319) to (102.75, 111.85, 20.1) mm, rotated rx 180 ry 0 rz -180 deg; joints [1.365, 65.936, -28.115, 2.226, -37.842, -1.758]
  Call Extruder 0.00932
  MoveL (T20320) to (111.05, 111.85, 20.1) mm, rotated rx 180 ry 0 rz -180 deg; joints [1.365, 65.936, -28.115, 2.226, -37.842, -1.758]
  Call Extruder 0.00013
  MoveL (T20321) to (111, 111.75, 20.1) mm, rotated rx 180 ry 0 rz -180 deg; joints [1.365, 65.936, -28.115, 2.226, -37.842, -1.758]
  Call Extruder 0.00926
  MoveL (T20322) to (102.75, 111.75, 20.1) mm, rotated rx 180 ry 0 rz -180 deg; joints [1.319, 71.114, -37.834, 2.404, -33.303, -2.009]
  Call Extruder 0.00011
  MoveL (T20323) to (102.75, 111.65, 20.1) mm, rotated rx 180 ry 0 rz -180 deg; joints [1.319, 71.114, -37.834, 2.404, -33.303, -2.009]
  Call Extruder 0.00921
  MoveL (T20324) to (110.95, 111.65, 20.1) mm, rotated rx 180 ry 0 rz -180 deg; joints [3.282, 71.353, -38.283, 5.998, -33.214, -5.024]
  Call Extruder 0.00013
  MoveL (T20325) to (110.9, 111.55, 20.1) mm, rotated rx 180 ry 0 rz -180 deg; joints [3.282, 71.353, -38.283, 5.998, -33.214, -5.024]
  Call Extruder 0.00915
  MoveL (T20326) to (102.75, 111.55, 20.1) mm, rotated rx 180 ry 0 rz -180 deg; joints [3.398, 66.034, -28.297, 5.541, -37.866, -4.379]
  Call Extruder 0.00011
  MoveL (T20327) to (102.75, 111.45, 20.1) mm, rotated rx 180 ry 0 rz -180 deg; joints [3.398, 66.034, -28.297, 5.541, -37.866, -4.379]
  Call Extruder 0.00909
  MoveL (T20328) to (110.85, 111.45, 20.1) mm, rotated rx 180 ry 0 rz -180 deg; joints [3.398, 66.034, -28.297, 5.541, -37.866, -4.379]
  Call Extruder 0.00013
  MoveL (T20329) to (110.8, 111.35, 20.1) mm, rotated rx 180 ry 0 rz -180 deg; joints [3.398, 66.034, -28.297, 5.541, -37.866, -4.379]
  Call Extruder 0.00903
  MoveL (T20330) to (102.75, 111.35, 20.1) mm, rotated rx 180 ry 0 rz -180 deg; joints [1.366, 65.834, -27.923, 2.223, -37.932, -1.754]
  Call Extruder 0.00011
  MoveL (T20331) to (102.75, 111.25, 20.1) mm, rotated rx 180 ry 0 rz -180 deg; joints [1.366, 65.834, -27.923, 2.223, -37.932, -1.754]
  Call Extruder 0.00898
  MoveL (T20332) to (110.75, 111.25, 20.1) mm, rotated rx 180 ry 0 rz -180 deg; joints [1.366, 65.834, -27.923, 2.223, -37.932, -1.754]
  Call Extruder 0.00013
  MoveL (T20333) to (110.7, 111.15, 20.1) mm, rotated rx 180 ry 0 rz -180 deg; joints [1.366, 65.834, -27.923, 2.223, -37.932, -1.754]
  Call Extruder 0.00892
  MoveL (T20334) to (102.75, 111.15, 20.1) mm, rotated rx 180 ry 0 rz -180 deg; joints [1.365, 65.921, -28.086, 2.225, -37.856, -1.757]
  Call Extruder 0.00011
  MoveL (T20335) to (102.75, 111.05, 20.1) mm, rotated rx 180 ry 0 rz -180 deg; joints [1.365, 65.921, -28.086, 2.225, -37.856, -1.757]
  Call Extruder 0.00886
  MoveL (T20336) to (110.64, 111.05, 20.1) mm, rotated rx 180 ry 0 rz -180 deg; joints [1.365, 65.921, -28.086, 2.225, -37.856, -1.757]
  Call Extruder 0.00013
  MoveL (T20337) to (110.59, 110.95, 20.1) mm, rotated rx 180 ry 0 rz -180 deg; joints [1.365, 65.921, -28.086, 2.225, -37.856, -1.757]
  Call Extruder 0.0088
  MoveL (T20338) to (102.75, 110.95, 20.1) mm, rotated rx 180 ry 0 rz -180 deg; joints [1.332, 65.729, -27.725, 2.163, -38.023, -1.705]
  Call Extruder 0.00011
  MoveL (T20339) to (102.75, 110.85, 20.1) mm, rotated rx 180 ry 0 rz -180 deg; joints [1.332, 65.729, -27.725, 2.163, -38.023, -1.705]
  Call Extruder 0.00875
  MoveL (T20340) to (110.54, 110.85, 20.1) mm, rotated rx 180 ry 0 rz -180 deg; joints [1.332, 65.729, -27.725, 2.163, -38.023, -1.705]
  Call Extruder 0.00013
  MoveL (T20341) to (110.49, 110.75, 20.1) mm, rotated rx 180 ry 0 rz -180 deg; joints [1.332, 65.729, -27.725, 2.163, -38.023, -1.705]
  Call Extruder 0.00869
  MoveL (T20342) to (102.75, 110.75, 20.1) mm, rotated rx 180 ry 0 rz -180 deg; joints [1.332, 65.729, -27.725, 2.163, -38.023, -1.705]
  Call Extruder 0.00011
  MoveL (T20343) to (102.75, 110.65, 20.1) mm, rotated rx 180 ry 0 rz -180 deg; joints [1.323, 65.728, -27.724, 2.148, -38.023, -1.693]
  Call Extruder 0.00863
  MoveL (T20344) to (110.44, 110.65, 20.1) mm, rotated rx 180 ry 0 rz -180 deg; joints [1.276, 71.24, -38.071, 2.331, -33.191, -1.951]
  Call Extruder 0.00013
  MoveL (T20345) to (110.39, 110.55, 20.1) mm, rotated rx 180 ry 0 rz -180 deg; joints [1.276, 71.24, -38.071, 2.331, -33.191, -1.951]
  Call Extruder 0.00858
  MoveL (T20346) to (102.75, 110.55, 20.1) mm, rotated rx 180 ry 0 rz -180 deg; joints [1.276, 71.24, -38.071, 2.331, -33.191, -1.951]
  Call Extruder 0.00011
  MoveL (T20347) to (102.75, 110.45, 20.1) mm, rotated rx 180 ry 0 rz -180 deg; joints [3.322, 71.49, -38.541, 6.091, -33.097, -5.108]
  Call Extruder 0.00852
  MoveL (T20348) to (110.34, 110.45, 20.1) mm, rotated rx 180 ry 0 rz -180 deg; joints [3.322, 71.49, -38.541, 6.091, -33.097, -5.108]
  Call Extruder 0.00013
  MoveL (T20349) to (110.29, 110.35, 20.1) mm, rotated rx 180 ry 0 rz -180 deg; joints [3.322, 71.49, -38.541, 6.091, -33.097, -5.108]
  Call Extruder 0.00846
  MoveL (T20350) to (102.75, 110.35, 20.1) mm, rotated rx 180 ry 0 rz -180 deg; joints [3.445, 65.936, -28.113, 5.606, -37.955, -4.426]
  Call Extruder 0.00011
  MoveL (T20351) to (102.75, 110.25, 20.1) mm, rotated rx 180 ry 0 rz -180 deg; joints [3.445, 65.936, -28.113, 5.606, -37.955, -4.426]
  Call Extruder 0.0084
  MoveL (T20352) to (110.24, 110.25, 20.1) mm, rotated rx 180 ry 0 rz -180 deg; joints [1.339, 65.729, -27.726, 2.174, -38.023, -1.713]
  Call Extruder 0.00013
  MoveL (T20353) to (110.19, 110.15, 20.1) mm, rotated rx 180 ry 0 rz -180 deg; joints [1.339, 65.729, -27.726, 2.174, -38.023, -1.713]
  Call Extruder 0.00835
  MoveL (T20354) to (102.75, 110.15, 20.1) mm, rotated rx 180 ry 0 rz -180 deg; joints [1.326, 65.744, -27.753, 2.153, -38.01, -1.697]
  Call Extruder 0.00011
  MoveL (T20355) to (102.75, 110.05, 20.1) mm, rotated rx 180 ry 0 rz -180 deg; joints [1.326, 65.744, -27.753, 2.153, -38.01, -1.697]
  Call Extruder 0.00829
  MoveL (T20356) to (110.14, 110.05, 20.1) mm, rotated rx 180 ry 0 rz -180 deg; joints [1.326, 65.744, -27.753, 2.153, -38.01, -1.697]
  Call Extruder 0.00013
  MoveL (T20357) to (110.08, 109.95, 20.1) mm, rotated rx 180 ry 0 rz -180 deg; joints [1.326, 65.744, -27.753, 2.153, -38.01, -1.697]
  Call Extruder 0.00823
  MoveL (T20358) to (102.75, 109.95, 20.1) mm, rotated rx 180 ry 0 rz -180 deg; joints [1.326, 65.744, -27.753, 2.153, -38.01, -1.697]
  Call Extruder 0.00011
  MoveL (T20359) to (102.75, 109.85, 20.1) mm, rotated rx 180 ry 0 rz -180 deg; joints [1.326, 65.744, -27.753, 2.153, -38.01, -1.697]
  Call Extruder 0.00817
  MoveL (T20360) to (110.03, 109.85, 20.1) mm, rotated rx 180 ry 0 rz -180 deg; joints [1.326, 65.744, -27.753, 2.153, -38.01, -1.697]
  Call Extruder 0.00013
  MoveL (T20361) to (109.98, 109.75, 20.1) mm, rotated rx 180 ry 0 rz -180 deg; joints [1.326, 65.744, -27.753, 2.153, -38.01, -1.697]
  Call Extruder 0.00812
  MoveL (T20362) to (102.75, 109.75, 20.1) mm, rotated rx 180 ry 0 rz -180 deg; joints [1.323, 65.728, -27.724, 2.148, -38.023, -1.693]
  Call Extruder 0.00011
  MoveL (T20363) to (102.75, 109.65, 20.1) mm, rotated rx 180 ry 0 rz -180 deg; joints [1.323, 65.728, -27.724, 2.148, -38.023, -1.693]
  Call Extruder 0.00806
  MoveL (T20364) to (109.93, 109.65, 20.1) mm, rotated rx 180 ry 0 rz -180 deg; joints [1.323, 65.728, -27.724, 2.148, -38.023, -1.693]
  Call Extruder 0.00013
  MoveL (T20365) to (109.88, 109.55, 20.1) mm, rotated rx 180 ry 0 rz -180 deg; joints [1.321, 65.963, -28.166, 2.155, -37.817, -1.702]
  Call Extruder 0.008
  MoveL (T20366) to (102.75, 109.55, 20.1) mm, rotated rx 180 ry 0 rz -180 deg; joints [1.321, 65.963, -28.166, 2.155, -37.817, -1.702]
  Call Extruder 0.00011
  MoveL (T20367) to (102.75, 109.45, 20.1) mm, rotated rx 180 ry 0 rz -180 deg; joints [1.321, 65.963, -28.166, 2.155, -37.817, -1.702]
  Call Extruder 0.00795
  MoveL (T20368) to (109.83, 109.45, 20.1) mm, rotated rx 180 ry 0 rz -180 deg; joints [1.321, 65.963, -28.166, 2.155, -37.817, -1.702]
  Call Extruder 0.00013
  MoveL (T20369) to (109.78, 109.35, 20.1) mm, rotated rx 180 ry 0 rz -180 deg; joints [1.321, 65.963, -28.166, 2.155, -37.817, -1.702]
  Call Extruder 0.00789
  MoveL (T20370) to (102.75, 109.35, 20.1) mm, rotated rx 180 ry 0 rz -180 deg; joints [1.321, 65.963, -28.166, 2.155, -37.817, -1.702]
  Call Extruder 0.00011
  MoveL (T20371) to (102.75, 109.25, 20.1) mm, rotated rx 180 ry 0 rz -180 deg; joints [1.707, 65.803, -28.271, 2.8, -37.565, -2.22]
  Call Extruder 0.00783
  MoveL (T20372) to (109.73, 109.25, 20.1) mm, rotated rx 180 ry 0 rz -180 deg; joints [1.707, 66.038, -28.306, 2.787, -37.765, -2.204]
  Call Extruder 0.00013
  MoveL (T20373) to (109.67, 109.15, 20.1) mm, rotated rx 180 ry 0 rz -180 deg; joints [1.707, 66.038, -28.306, 2.787, -37.765, -2.204]
  Call Extruder 0.00777
  MoveL (T20374) to (102.75, 109.15, 20.1) mm, rotated rx 180 ry 0 rz -180 deg; joints [1.707, 66.038, -28.306, 2.787, -37.765, -2.204]
  Call Extruder 0.00011
  MoveL (T20375) to (102.75, 109.05, 20.1) mm, rotated rx 180 ry 0 rz -180 deg; joints [1.707, 66.038, -28.306, 2.787, -37.765, -2.204]
  Call Extruder 0.00772
  MoveL (T20376) to (109.62, 109.05, 20.1) mm, rotated rx 180 ry 0 rz -180 deg; joints [1.707, 66.038, -28.306, 2.787, -37.765, -2.204]
  Call Extruder 0.00013
  MoveL (T20377) to (109.57, 108.95, 20.1) mm, rotated rx 180 ry 0 rz -180 deg; joints [1.707, 66.038, -28.306, 2.787, -37.765, -2.204]
  Call Extruder 0.00766
  MoveL (T20378) to (102.75, 108.95, 20.1) mm, rotated rx 180 ry 0 rz -180 deg; joints [1.707, 66.038, -28.306, 2.787, -37.765, -2.204]
  Call Extruder 0.00011
  MoveL (T20379) to (102.75, 108.85, 20.1) mm, rotated rx 180 ry 0 rz -180 deg; joints [1.707, 66.038, -28.306, 2.787, -37.765, -2.204]
  Call Extruder 0.0076
  MoveL (T20380) to (109.52, 108.85, 20.1) mm, rotated rx 180 ry 0 rz -180 deg; joints [1.442, 66.021, -28.273, 2.354, -37.771, -1.861]
  Call Extruder 0.00013
  MoveL (T20381) to (109.47, 108.75, 20.1) mm, rotated rx 180 ry 0 rz -180 deg; joints [1.442, 66.021, -28.273, 2.354, -37.771, -1.861]
  Call Extruder 0.00754
  MoveL (T20382) to (102.75, 108.75, 20.1) mm, rotated rx 180 ry 0 rz -180 deg; joints [1.501, 66.169, -28.551, 2.458, -37.644, -1.947]
  Call Extruder 0.00011
  MoveL (T20383) to (102.75, 108.65, 20.1) mm, rotated rx 180 ry 0 rz -180 deg; joints [1.501, 66.169, -28.551, 2.458, -37.644, -1.947]
  Call Extruder 0.00749
  MoveL (T20384) to (109.42, 108.65, 20.1) mm, rotated rx 180 ry 0 rz -180 deg; joints [1.501, 66.169, -28.551, 2.458, -37.644, -1.947]
  Call Extruder 0.00013
  MoveL (T20385) to (109.37, 108.55, 20.1) mm, rotated rx 180 ry 0 rz -180 deg; joints [1.643, 66.178, -28.568, 2.691, -37.64, -2.132]
  Call Extruder 0.00743
  MoveL (T20386) to (102.75, 108.55, 20.1) mm, rotated rx 180 ry 0 rz -180 deg; joints [1.643, 66.178, -28.568, 2.691, -37.64, -2.132]
  Call Extruder 0.00011
  MoveL (T20387) to (102.75, 108.45, 20.1) mm, rotated rx 180 ry 0 rz -180 deg; joints [1.643, 66.178, -28.568, 2.691, -37.64, -2.132]
  Call Extruder 0.00737
  MoveL (T20388) to (109.32, 108.45, 20.1) mm, rotated rx 180 ry 0 rz -180 deg; joints [1.699, 66.319, -28.833, 2.79, -37.519, -2.214]
  Call Extruder 0.00013
  MoveL (T20389) to (109.27, 108.35, 20.1) mm, rotated rx 180 ry 0 rz -180 deg; joints [1.699, 66.319, -28.833, 2.79, -37.519, -2.214]
  Call Extruder 0.00732
  MoveL (T20390) to (102.75, 108.35, 20.1) mm, rotated rx 180 ry 0 rz -180 deg; joints [1.821, 66.046, -28.321, 2.974, -37.763, -2.352]
  Call Extruder 0.00011
  MoveL (T20391) to (102.75, 108.25, 20.1) mm, rotated rx 180 ry 0 rz -180 deg; joints [1.941, 66.056, -28.339, 3.171, -37.759, -2.508]
  Call Extruder 0.00726
  MoveL (T20392) to (109.22, 108.25, 20.1) mm, rotated rx 180 ry 0 rz -180 deg; joints [1.941, 66.056, -28.339, 3.171, -37.759, -2.508]
  Call Extruder 0.00013
  MoveL (T20393) to (109.17, 108.15, 20.1) mm, rotated rx 180 ry 0 rz -180 deg; joints [3.239, 69.708, -35.194, 5.703, -34.647, -4.697]
  Call Extruder 0.0072
  MoveL (T20394) to (102.75, 108.15, 20.1) mm, rotated rx 180 ry 0 rz -180 deg; joints [3.232, 70.039, -35.816, 5.733, -34.357, -4.738]
  Call Extruder 0.00011
  MoveL (T20395) to (102.75, 108.05, 20.1) mm, rotated rx 180 ry 0 rz -180 deg; joints [3.232, 70.039, -35.816, 5.733, -34.357, -4.738]
  Call Extruder 0.00714
  MoveL (T20396) to (109.11, 108.05, 20.1) mm, rotated rx 180 ry 0 rz -180 deg; joints [2.845, 71.056, -37.726, 5.168, -33.438, -4.316]
  Call Extruder 0.00013
  MoveL (T20397) to (109.06, 107.95, 20.1) mm, rotated rx 180 ry 0 rz -180 deg; joints [2.845, 71.056, -37.726, 5.168, -33.438, -4.316]
  Call Extruder 0.00709
  MoveL (T20398) to (102.75, 107.95, 20.1) mm, rotated rx 180 ry 0 rz -180 deg; joints [2.729, 71.039, -37.694, 4.956, -33.444, -4.138]
  Call Extruder 0.00011
  MoveL (T20399) to (102.75, 107.85, 20.1) mm, rotated rx 180 ry 0 rz -180 deg; joints [2.729, 71.039, -37.694, 4.956, -33.444, -4.138]
  Call Extruder 0.00703
  MoveL (T20400) to (109.01, 107.85, 20.1) mm, rotated rx 180 ry 0 rz -180 deg; joints [2.695, 70.928, -37.485, 4.882, -33.539, -4.072]
  Call Extruder 0.00013
  MoveL (T20401) to (108.96, 107.75, 20.1) mm, rotated rx 180 ry 0 rz -180 deg; joints [2.703, 70.436, -36.561, 4.841, -33.97, -4.018]
  Call Extruder 0.00697
  MoveL (T20402) to (102.75, 107.75, 20.1) mm, rotated rx 180 ry 0 rz -180 deg; joints [2.703, 70.436, -36.561, 4.841, -33.97, -4.018]
  Call Extruder 0.00011
  MoveL (T20403) to (102.75, 107.65, 20.1) mm, rotated rx 180 ry 0 rz -180 deg; joints [2.703, 70.436, -36.561, 4.841, -33.97, -4.018]
  Call Extruder 0.00692
  MoveL (T20404) to (108.91, 107.65, 20.1) mm, rotated rx 180 ry 0 rz -180 deg; joints [2.641, 70.241, -36.194, 4.71, -34.137, -3.902]
  Call Extruder 0.00013
  MoveL (T20405) to (108.86, 107.55, 20.1) mm, rotated rx 180 ry 0 rz -180 deg; joints [3.26, 68.696, -33.293, 5.615, -35.533, -4.574]
  Call Extruder 0.00686
  MoveL (T20406) to (102.75, 107.55, 20.1) mm, rotated rx 180 ry 0 rz -180 deg; joints [3.26, 68.696, -33.293, 5.615, -35.533, -4.574]
  Call Extruder 0.00011
  MoveL (T20407) to (102.75, 107.45, 20.1) mm, rotated rx 180 ry 0 rz -180 deg; joints [3.266, 68.382, -32.704, 5.589, -35.807, -4.537]
  Call Extruder 0.0068
  MoveL (T20408) to (108.81, 107.45, 20.1) mm, rotated rx 180 ry 0 rz -180 deg; joints [2.44, 66.101, -28.424, 3.988, -37.744, -3.155]
  Call Extruder 0.00013
  MoveL (T20409) to (108.76, 107.35, 20.1) mm, rotated rx 180 ry 0 rz -180 deg; joints [2.44, 66.101, -28.424, 3.988, -37.744, -3.155]
  Call Extruder 0.00674
  MoveL (T20410) to (102.75, 107.35, 20.1) mm, rotated rx 180 ry 0 rz -180 deg; joints [2.319, 66.089, -28.401, 3.79, -37.748, -2.999]
  Call Extruder 0.00011
  MoveL (T20411) to (102.75, 107.25, 20.1) mm, rotated rx 180 ry 0 rz -180 deg; joints [2.319, 66.089, -28.401, 3.79, -37.748, -2.999]
  Call Extruder 0.00669
  MoveL (T20412) to (108.71, 107.25, 20.1) mm, rotated rx 180 ry 0 rz -180 deg; joints [1.833, 67.189, -30.465, 3.064, -36.763, -2.455]
  Call Extruder 0.00013
  MoveL (T20413) to (108.66, 107.15, 20.1) mm, rotated rx 180 ry 0 rz -180 deg; joints [1.833, 67.189, -30.465, 3.064, -36.763, -2.455]
  Call Extruder 0.00663
  MoveL (T20414) to (102.75, 107.15, 20.1) mm, rotated rx 180 ry 0 rz -180 deg; joints [1.833, 67.189, -30.465, 3.064, -36.763, -2.455]
  Call Extruder 0.00011
  MoveL (T20415) to (102.75, 107.05, 20.1) mm, rotated rx 180 ry 0 rz -180 deg; joints [1.835, 67.029, -30.165, 3.057, -36.903, -2.446]
  Call Extruder 0.00657
  MoveL (T20416) to (108.6, 107.05, 20.1) mm, rotated rx 180 ry 0 rz -180 deg; joints [3.211, 71.114, -37.835, 5.838, -33.416, -4.878]
  Call Extruder 0.00012
  MoveL (T20417) to (108.57, 106.95, 20.1) mm, rotated rx 180 ry 0 rz -180 deg; joints [3.211, 71.114, -37.835, 5.838, -33.416, -4.878]
  Call Extruder 0.00654
  MoveL (T20418) to (102.75, 106.95, 20.1) mm, rotated rx 180 ry 0 rz -180 deg; joints [3.226, 70.358, -36.414, 5.763, -34.079, -4.779]
  Call Extruder 0.00011
  MoveL (T20419) to (102.75, 106.85, 20.1) mm, rotated rx 180 ry 0 rz -180 deg; joints [3.226, 70.358, -36.414, 5.763, -34.079, -4.779]
  Call Extruder 0.00654
  MoveL (T20420) to (108.57, 106.85, 20.1) mm, rotated rx 180 ry 0 rz -180 deg; joints [3.226, 70.358, -36.414, 5.763, -34.079, -4.779]
  Call Extruder 0.00011
  MoveL (T20421) to (108.57, 106.75, 20.1) mm, rotated rx 180 ry 0 rz -180 deg; joints [3.226, 70.358, -36.414, 5.763, -34.079, -4.779]
  Call Extruder 0.00654
  MoveL (T20422) to (102.75, 106.75, 20.1) mm, rotated rx 180 ry 0 rz -180 deg; joints [3.226, 70.358, -36.414, 5.763, -34.079, -4.779]
  Call Extruder 0.00011
  MoveL (T20423) to (102.75, 106.65, 20.1) mm, rotated rx 180 ry 0 rz -180 deg; joints [3.226, 70.358, -36.414, 5.763, -34.079, -4.779]
  Call Extruder 0.00654
  MoveL (T20424) to (108.57, 106.65, 20.1) mm, rotated rx 180 ry 0 rz -180 deg; joints [3.226, 70.358, -36.414, 5.763, -34.079, -4.779]
  Call Extruder 0.00011
  MoveL (T20425) to (108.57, 106.55, 20.1) mm, rotated rx 180 ry 0 rz -180 deg; joints [3.219, 70.685, -37.028, 5.795, -33.792, -4.821]
  Call Extruder 0.00654
  MoveL (T20426) to (102.75, 106.55, 20.1) mm, rotated rx 180 ry 0 rz -180 deg; joints [3.219, 70.685, -37.028, 5.795, -33.792, -4.821]
  Call Extruder 0.00011
  MoveL (T20427) to (102.75, 106.45, 20.1) mm, rotated rx 180 ry 0 rz -180 deg; joints [3.219, 70.685, -37.028, 5.795, -33.792, -4.821]
  Call Extruder 0.00654
  MoveL (T20428) to (108.57, 106.45, 20.1) mm, rotated rx 180 ry 0 rz -180 deg; joints [3.219, 70.685, -37.028, 5.795, -33.792, -4.821]
  Call Extruder 0.00011
  MoveL (T20429) to (108.57, 106.35, 20.1) mm, rotated rx 180 ry 0 rz -180 deg; joints [3.219, 70.453, -36.988, 5.824, -33.601, -4.856]
  Call Extruder 0.00654
  MoveL (T20430) to (102.75, 106.35, 20.1) mm, rotated rx 180 ry 0 rz -180 deg; joints [2.593, 70.847, -37.727, 4.737, -33.21, -3.966]
  Call Extruder 0.00011
  MoveL (T20431) to (102.75, 106.25, 20.1) mm, rotated rx 180 ry 0 rz -180 deg; joints [2.593, 70.847, -37.727, 4.737, -33.21, -3.966]
  Call Extruder 0.02189
  MoveL (T20432) to (122.25, 106.25, 20.1) mm, rotated rx 180 ry 0 rz -180 deg; joints [2.593, 71.078, -37.768, 4.713, -33.4, -3.938]
  Call Extruder 0.00011
  MoveL (T20433) to (122.25, 106.15, 20.1) mm, rotated rx 180 ry 0 rz -180 deg; joints [2.593, 71.078, -37.768, 4.713, -33.4, -3.938]
  Call Extruder 0.02189
  MoveL (T20434) to (102.75, 106.15, 20.1) mm, rotated rx 180 ry 0 rz -180 deg; joints [2.593, 71.078, -37.768, 4.713, -33.4, -3.938]
  Call Extruder 0.00011
  MoveL (T20435) to (102.75, 106.05, 20.1) mm, rotated rx 180 ry 0 rz -180 deg; joints [2.593, 71.078, -37.768, 4.713, -33.4, -3.938]
  Call Extruder 0.02189
  MoveL (T20436) to (122.25, 106.05, 20.1) mm, rotated rx 180 ry 0 rz -180 deg; joints [2.593, 71.078, -37.768, 4.713, -33.4, -3.938]
  Call Extruder 0.00011
  MoveL (T20437) to (122.25, 105.95, 20.1) mm, rotated rx 180 ry 0 rz -180 deg; joints [2.593, 71.078, -37.768, 4.713, -33.4, -3.938]
  Call Extruder 0.02189
  MoveL (T20438) to (102.75, 105.95, 20.1) mm, rotated rx 180 ry 0 rz -180 deg; joints [2.655, 70.908, -37.447, 4.808, -33.554, -4.009]
  Call Extruder 0.00011
  MoveL (T20439) to (102.75, 105.85, 20.1) mm, rotated rx 180 ry 0 rz -180 deg; joints [2.658, 70.748, -37.147, 4.795, -33.693, -3.992]
  Call Extruder 0.02189
  MoveL (T20440) to (122.25, 105.85, 20.1) mm, rotated rx 180 ry 0 rz -180 deg; joints [2.658, 70.748, -37.147, 4.795, -33.693, -3.992]
  Call Extruder 0.00011
  MoveL (T20441) to (122.25, 105.75, 20.1) mm, rotated rx 180 ry 0 rz -180 deg; joints [2.557, 71.023, -37.664, 4.642, -33.446, -3.876]
  Call Extruder 0.02189
  MoveL (T20442) to (102.75, 105.75, 20.1) mm, rotated rx 180 ry 0 rz -180 deg; joints [2.557, 71.023, -37.664, 4.642, -33.446, -3.876]
  Call Extruder 0.00011
  MoveL (T20443) to (102.75, 105.65, 20.1) mm, rotated rx 180 ry 0 rz -180 deg; joints [2.557, 71.023, -37.664, 4.642, -33.446, -3.876]
  Call Extruder 0.02189
  MoveL (T20444) to (122.25, 105.65, 20.1) mm, rotated rx 180 ry 0 rz -180 deg; joints [2.503, 71.016, -37.65, 4.544, -33.449, -3.794]
  Call Extruder 0.00011
  MoveL (T20445) to (122.25, 105.55, 20.1) mm, rotated rx 180 ry 0 rz -180 deg; joints [2.66, 70.59, -36.85, 4.782, -33.832, -3.975]
  Call Extruder 0.02189
  MoveL (T20446) to (102.75, 105.55, 20.1) mm, rotated rx 180 ry 0 rz -180 deg; joints [2.66, 70.59, -36.85, 4.782, -33.832, -3.975]
  Call Extruder 0.00011
  MoveL (T20447) to (102.75, 105.45, 20.1) mm, rotated rx 180 ry 0 rz -180 deg; joints [2.66, 70.59, -36.85, 4.782, -33.832, -3.975]
  Call Extruder 0.02189
  MoveL (T20448) to (122.25, 105.45, 20.1) mm, rotated rx 180 ry 0 rz -180 deg; joints [2.662, 70.479, -36.642, 4.773, -33.929, -3.963]
  Call Extruder 0.00011
  MoveL (T20449) to (122.25, 105.35, 20.1) mm, rotated rx 180 ry 0 rz -180 deg; joints [2.662, 70.479, -36.642, 4.773, -33.929, -3.963]
  Call Extruder 0.02189
  MoveL (T20450) to (102.75, 105.35, 20.1) mm, rotated rx 180 ry 0 rz -180 deg; joints [2.662, 70.479, -36.642, 4.773, -33.929, -3.963]
  Call Extruder 0.00011
  MoveL (T20451) to (102.75, 105.25, 20.1) mm, rotated rx 180 ry 0 rz -180 deg; joints [2.654, 70.455, -36.596, 4.757, -33.95, -3.949]
  Call Extruder 0.02189
  MoveL (T20452) to (122.25, 105.25, 20.1) mm, rotated rx 180 ry 0 rz -180 deg; joints [2.449, 71.009, -37.637, 4.446, -33.451, -3.712]
  Call Extruder 0.00011
  MoveL (T20453) to (122.25, 105.15, 20.1) mm, rotated rx 180 ry 0 rz -180 deg; joints [2.449, 71.009, -37.637, 4.446, -33.451, -3.712]
  Call Extruder 0.02189
  MoveL (T20454) to (102.75, 105.15, 20.1) mm, rotated rx 180 ry 0 rz -180 deg; joints [2.395, 71.002, -37.625, 4.348, -33.454, -3.63]
  Call Extruder 0.00011
  MoveL (T20455) to (102.75, 105.05, 20.1) mm, rotated rx 180 ry 0 rz -180 deg; joints [2.629, 70.373, -36.443, 4.702, -34.02, -3.9]
  Call Extruder 0.02189
  MoveL (T20456) to (122.25, 105.05, 20.1) mm, rotated rx 180 ry 0 rz -180 deg; joints [2.629, 70.373, -36.443, 4.702, -34.02, -3.9]
  Call Extruder 0.00011
  MoveL (T20457) to (122.25, 104.95, 20.1) mm, rotated rx 180 ry 0 rz -180 deg; joints [2.629, 70.373, -36.443, 4.702, -34.02, -3.9]
  Call Extruder 0.02189
  MoveL (T20458) to (102.75, 104.95, 20.1) mm, rotated rx 180 ry 0 rz -180 deg; joints [2.603, 70.292, -36.29, 4.648, -34.089, -3.852]
  Call Extruder 0.00011
  MoveL (T20459) to (102.75, 104.85, 20.1) mm, rotated rx 180 ry 0 rz -180 deg; joints [2.603, 70.292, -36.29, 4.648, -34.089, -3.852]
  Call Extruder 0.02189
  MoveL (T20460) to (122.25, 104.85, 20.1) mm, rotated rx 180 ry 0 rz -180 deg; joints [2.342, 70.996, -37.612, 4.25, -33.456, -3.548]
  Call Extruder 0.00011
  MoveL (T20461) to (122.25, 104.75, 20.1) mm, rotated rx 180 ry 0 rz -180 deg; joints [2.342, 70.996, -37.612, 4.25, -33.456, -3.548]
  Call Extruder 0.02189
  MoveL (T20462) to (102.75, 104.75, 20.1) mm, rotated rx 180 ry 0 rz -180 deg; joints [2.342, 70.996, -37.612, 4.25, -33.456, -3.548]
  Call Extruder 0.00011
  MoveL (T20463) to (102.75, 104.65, 20.1) mm, rotated rx 180 ry 0 rz -180 deg; joints [2.288, 70.989, -37.6, 4.153, -33.459, -3.466]
  Call Extruder 0.02189
  MoveL (T20464) to (122.25, 104.65, 20.1) mm, rotated rx 180 ry 0 rz -180 deg; joints [2.288, 70.989, -37.6, 4.153, -33.459, -3.466]
  Call Extruder 0.00011
  MoveL (T20465) to (122.25, 104.55, 20.1) mm, rotated rx 180 ry 0 rz -180 deg; joints [2.577, 70.21, -36.137, 4.593, -34.159, -3.803]
  Call Extruder 0.02189
  MoveL (T20466) to (102.75, 104.55, 20.1) mm, rotated rx 180 ry 0 rz -180 deg; joints [2.577, 70.21, -36.137, 4.593, -34.159, -3.803]
  Call Extruder 0.00011
  MoveL (T20467) to (102.75, 104.45, 20.1) mm, rotated rx 180 ry 0 rz -180 deg; joints [2.551, 70.13, -35.986, 4.539, -34.228, -3.756]
  Call Extruder 0.02189
  MoveL (T20468) to (122.25, 104.45, 20.1) mm, rotated rx 180 ry 0 rz -180 deg; joints [2.234, 70.983, -37.588, 4.055, -33.461, -3.384]
  Call Extruder 0.00011
  MoveL (T20469) to (122.25, 104.35, 20.1) mm, rotated rx 180 ry 0 rz -180 deg; joints [2.181, 70.977, -37.576, 3.957, -33.463, -3.303]
  Call Extruder 0.02189
  MoveL (T20470) to (102.75, 104.35, 20.1) mm, rotated rx 180 ry 0 rz -180 deg; joints [2.181, 70.977, -37.576, 3.957, -33.463, -3.303]
  Call Extruder 0.00011
  MoveL (T20471) to (102.75, 104.25, 20.1) mm, rotated rx 180 ry 0 rz -180 deg; joints [2.181, 70.977, -37.576, 3.957, -33.463, -3.303]
  Call Extruder 0.02189
  MoveL (T20472) to (122.25, 104.25, 20.1) mm, rotated rx 180 ry 0 rz -180 deg; joints [2.526, 70.049, -35.835, 4.485, -34.296, -3.708]
  Call Extruder 0.00011
  MoveL (T20473) to (122.25, 104.15, 20.1) mm, rotated rx 180 ry 0 rz -180 deg; joints [2.5, 69.969, -35.684, 4.432, -34.365, -3.66]
  Call Extruder 0.02189
  MoveL (T20474) to (102.75, 104.15, 20.1) mm, rotated rx 180 ry 0 rz -180 deg; joints [2.127, 70.971, -37.565, 3.859, -33.465, -3.221]
  Call Extruder 0.00011
  MoveL (T20475) to (102.75, 104.05, 20.1) mm, rotated rx 180 ry 0 rz -180 deg; joints [2.127, 70.971, -37.565, 3.859, -33.465, -3.221]
  Call Extruder 0.02189
  MoveL (T20476) to (122.25, 104.05, 20.1) mm, rotated rx 180 ry 0 rz -180 deg; joints [2.073, 70.965, -37.554, 3.761, -33.468, -3.139]
  Call Extruder 0.00011
  MoveL (T20477) to (122.25, 103.95, 20.1) mm, rotated rx 180 ry 0 rz -180 deg; joints [2.073, 70.965, -37.554, 3.761, -33.468, -3.139]
  Call Extruder 0.02189
  MoveL (T20478) to (102.75, 103.95, 20.1) mm, rotated rx 180 ry 0 rz -180 deg; joints [2.45, 69.951, -35.649, 4.343, -34.378, -3.586]
  Call Extruder 0.00011
  MoveL (T20479) to (102.75, 103.85, 20.1) mm, rotated rx 180 ry 0 rz -180 deg; joints [2.396, 69.944, -35.637, 4.246, -34.38, -3.506]
  Call Extruder 0.02189
  MoveL (T20480) to (122.25, 103.85, 20.1) mm, rotated rx 180 ry 0 rz -180 deg; joints [2.02, 70.959, -37.543, 3.664, -33.47, -3.057]
  Call Extruder 0.00011
  MoveL (T20481) to (122.25, 103.75, 20.1) mm, rotated rx 180 ry 0 rz -180 deg; joints [2.02, 70.959, -37.543, 3.664, -33.47, -3.057]
  Call Extruder 0.02189
  MoveL (T20482) to (102.75, 103.75, 20.1) mm, rotated rx 180 ry 0 rz -180 deg; joints [2.02, 70.959, -37.543, 3.664, -33.47, -3.057]
  Call Extruder 0.00011
  MoveL (T20483) to (102.75, 103.65, 20.1) mm, rotated rx 180 ry 0 rz -180 deg; joints [1.966, 70.953, -37.533, 3.566, -33.472, -2.976]
  Call Extruder 0.02189
  MoveL (T20484) to (122.25, 103.65, 20.1) mm, rotated rx 180 ry 0 rz -180 deg; joints [2.342, 69.938, -35.626, 4.15, -34.382, -3.427]
  Call Extruder 0.00011
  MoveL (T20485) to (122.25, 103.55, 20.1) mm, rotated rx 180 ry 0 rz -180 deg; joints [2.342, 69.938, -35.626, 4.15, -34.382, -3.427]
  Call Extruder 0.02189
  MoveL (T20486) to (102.75, 103.55, 20.1) mm, rotated rx 180 ry 0 rz -180 deg; joints [2.288, 69.932, -35.614, 4.054, -34.385, -3.347]
  Call Extruder 0.00011
  MoveL (T20487) to (102.75, 103.45, 20.1) mm, rotated rx 180 ry 0 rz -180 deg; joints [2.288, 69.932, -35.614, 4.054, -34.385, -3.347]
  Call Extruder 0.02189
  MoveL (T20488) to (122.25, 103.45, 20.1) mm, rotated rx 180 ry 0 rz -180 deg; joints [1.912, 70.948, -37.523, 3.468, -33.474, -2.894]
  Call Extruder 0.00011
  MoveL (T20489) to (122.25, 103.35, 20.1) mm, rotated rx 180 ry 0 rz -180 deg; joints [1.885, 70.945, -37.518, 3.419, -33.475, -2.853]
  Call Extruder 0.02189
  MoveL (T20490) to (102.75, 103.35, 20.1) mm, rotated rx 180 ry 0 rz -180 deg; joints [1.885, 70.945, -37.518, 3.419, -33.475, -2.853]
  Call Extruder 0.00011
  MoveL (T20491) to (102.75, 103.25, 20.1) mm, rotated rx 180 ry 0 rz -180 deg; joints [1.885, 70.945, -37.518, 3.419, -33.475, -2.853]
  Call Extruder 0.02189
  MoveL (T20492) to (122.25, 103.25, 20.1) mm, rotated rx 180 ry 0 rz -180 deg; joints [1.885, 70.945, -37.518, 3.419, -33.475, -2.853]
  Call Extruder 0.00011
  MoveL (T20493) to (122.25, 103.15, 20.1) mm, rotated rx 180 ry 0 rz -180 deg; joints [2.234, 69.926, -35.603, 3.958, -34.387, -3.268]
  Call Extruder 0.02189
  MoveL (T20494) to (102.75, 103.15, 20.1) mm, rotated rx 180 ry 0 rz -180 deg; joints [2.18, 69.92, -35.592, 3.862, -34.389, -3.188]
  Call Extruder 0.00011
  MoveL (T20495) to (102.75, 103.05, 20.1) mm, rotated rx 180 ry 0 rz -180 deg; joints [2.18, 69.92, -35.592, 3.862, -34.389, -3.188]
  Call Extruder 0.02189
  MoveL (T20496) to (122.25, 103.05, 20.1) mm, rotated rx 180 ry 0 rz -180 deg; joints [1.888, 70.706, -37.069, 3.405, -33.684, -2.835]
  Call Extruder 0.00011
  MoveL (T20497) to (122.25, 102.95, 20.1) mm, rotated rx 180 ry 0 rz -180 deg; joints [1.89, 70.548, -36.772, 3.396, -33.823, -2.822]
  Call Extruder 0.02189
  MoveL (T20498) to (102.75, 102.95, 20.1) mm, rotated rx 180 ry 0 rz -180 deg; joints [1.89, 70.548, -36.772, 3.396, -33.823, -2.822]
  Call Extruder 0.00011
  MoveL (T20499) to (102.75, 102.85, 20.1) mm, rotated rx 180 ry 0 rz -180 deg; joints [2.126, 69.914, -35.581, 3.766, -34.391, -3.109]
  Call Extruder 0.02194
  MoveL (T20500) to (122.3, 102.85, 20.1) mm, rotated rx 180 ry 0 rz -180 deg; joints [2.126, 69.914, -35.581, 3.766, -34.391, -3.109]
  Set speed (45.0 mm/s)
  Call Extruder -1.6
  MoveL (T20501) to (122.3, 102.85, 20.1) mm, rotated rx 180 ry 0 rz -180 deg; joints [2.072, 69.909, -35.571, 3.67, -34.393, -3.03]
  Set speed (120.0 mm/s)
  MoveL (T20502) to (122.3, 102.85, 20.1) mm, rotated rx 180 ry 0 rz -180 deg; joints [1.874, 70.439, -36.567, 3.36, -33.918, -2.789]
  Call Extruder -0.38
  MoveL (T20503) to (121.23, 102.85, 20.1) mm, rotated rx 180 ry 0 rz -180 deg; joints [1.874, 70.439, -36.567, 3.36, -33.918, -2.789]
  Set speed (45.0 mm/s)
  Call Extruder -0.02
  MoveL (T20504) to (121.23, 102.85, 20.1) mm, rotated rx 180 ry 0 rz -180 deg; joints [1.874, 70.439, -36.567, 3.36, -33.918, -2.789]
  Set speed (150.0 mm/s)
  MoveL (T20505) to (121.23, 102.85, 22.1) mm, rotated rx 180 ry 0 rz -180 deg; joints [1.874, 70.439, -36.567, 3.36, -33.918, -2.789]
  Call Mcode M107
  MoveL (T20506) to (121.23, 102.85, 22.1) mm, rotated rx 180 ry 0 rz -180 deg; joints [1.874, 70.439, -36.567, 3.36, -33.918, -2.789]
